{attribute 'qualified_only'}
{attribute 'strict'}
TYPE E_VisionState :
(
	Idle := 0,
	SelectMode,
	Configure,
	Acquisition,
	Error
);
END_TYPE

(* stored: Version 1.1.0.1, ProductVersion 3.1.4024.13
   DUT E_VisionState: Id {37a6ed51-c96e-498f-ab82-bbd991d054c6} *)
